INTERFACE ITF_ExecuteFB

METHOD METH_Execute : BOOL
VAR_INPUT
END_VAR
END_METHOD

PROPERTY Prop_Execute : BOOL
GET
END_GET
SET
END_SET
END_PROPERTY

END_INTERFACE

(* stored: Version 1.1.0.1, ProductVersion 3.1.4024.12
   Itf ITF_ExecuteFB: Id {5706ecae-6e8b-40f4-b4de-659a4ea8d3a8}
   Method METH_Execute: Id {032595a5-0ec5-4ba7-87b3-5513c62ea9dc}
   Property Prop_Execute: Id {ed214682-318d-46e0-a0a5-b306cfe2d2d8}
   Get Get: Id {4c5191d0-9807-486a-b893-509ca0b5edca}
   Set Set: Id {a7396123-fe8d-48f3-b816-d8d768e39004} *)
